// TIA Portal project "Project_ToggleButton" (V16)

(* hardware
DEVICE "S7-1200 station_1"  S7-1200 Station
   slot 0: "Rack_0"  S7-1200 Rack  Rack  V1.0
   slot 1: "PLC_1"  CPU 1212C DC/DC/Rly  6ES7 212-1HE40-0XB0  V4.4
*)

// ===== PLC "PLC_1"  CPU 1212C DC/DC/Rly =====

VAR_GLOBAL   // PLC tag table "Default tag table"
   "TOGGLE BUTON" AT %I0.0 : Bool;
   "M1" AT %M50.0 : Bool;
   "M2" AT %M50.1 : Bool;
   "M3" AT %M50.2 : Bool;
   "M4" AT %M50.3 : Bool;
   "CIKIS" AT %Q0.0 : Bool;
END_VAR

ORGANIZATION_BLOCK "Main"   // OB1, LAD, ProgramCycle
TITLE = "Main Program Sweep (Cycle)"
{ S7_Optimized_Access := 'TRUE' }
VERSION : 0.1
   VAR_INPUT
      Initial_Call : Bool;   // Initial call of this OB
      Remanence : Bool;   // =True, if remanent data are available
   END_VAR
BEGIN

REGION Network 1: BUTONA 1.KEZ BASILDI
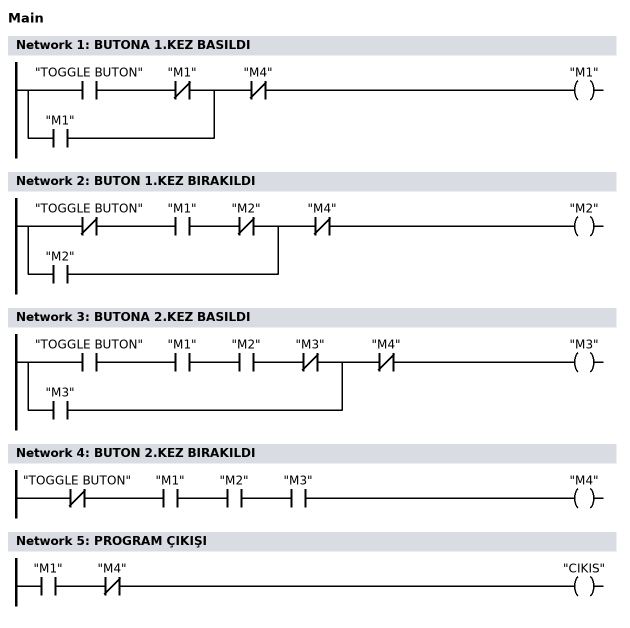
   RUNG wire#powerrail
      Contact( "TOGGLE BUTON" )
      I_Contact( "M1" )
      wire#w1
      I_Contact( "M4" )
      Coil( "M1" )
   END_RUNG
   RUNG wire#powerrail
      Contact( "M1" )
   END_RUNG wire#w1
   // the same network as SCL:
   "M1" := (("TOGGLE BUTON" AND NOT "M1") OR "M1") AND NOT "M4";
END_REGION

REGION Network 2: BUTON 1.KEZ BIRAKILDI
   RUNG wire#powerrail
      I_Contact( "TOGGLE BUTON" )
      Contact( "M1" )
      I_Contact( "M2" )
      wire#w1
      I_Contact( "M4" )
      Coil( "M2" )
   END_RUNG
   RUNG wire#powerrail
      Contact( "M2" )
   END_RUNG wire#w1
   // the same network as SCL:
   "M2" := ((NOT "TOGGLE BUTON" AND "M1" AND NOT "M2") OR "M2") AND NOT "M4";
END_REGION

REGION Network 3: BUTONA 2.KEZ BASILDI
   RUNG wire#powerrail
      Contact( "TOGGLE BUTON" )
      Contact( "M1" )
      Contact( "M2" )
      I_Contact( "M3" )
      wire#w1
      I_Contact( "M4" )
      Coil( "M3" )
   END_RUNG
   RUNG wire#powerrail
      Contact( "M3" )
   END_RUNG wire#w1
   // the same network as SCL:
   "M3" := (("TOGGLE BUTON" AND "M1" AND "M2" AND NOT "M3") OR "M3") AND NOT "M4";
END_REGION

REGION Network 4: BUTON 2.KEZ BIRAKILDI
   RUNG wire#powerrail
      I_Contact( "TOGGLE BUTON" )
      Contact( "M1" )
      Contact( "M2" )
      Contact( "M3" )
      Coil( "M4" )
   END_RUNG
   // the same network as SCL:
   "M4" := NOT "TOGGLE BUTON" AND "M1" AND "M2" AND "M3";
END_REGION

REGION Network 5: PROGRAM ÇIKIŞI
   RUNG wire#powerrail
      Contact( "M1" )
      I_Contact( "M4" )
      Coil( "CIKIS" )
   END_RUNG
   // the same network as SCL:
   "CIKIS" := "M1" AND NOT "M4";
END_REGION
END_ORGANIZATION_BLOCK